{attribute 'GeneratedUsingTerminal: EL6002-0000-0019'}
{attribute addProperty BoxType "EL6002-0000-0019"}
{attribute addProperty Id "StatusAT %I*Status_3D84275F8Data_InAT %I*ARRAY[0..21] OF USINT22"}
{attribute addProperty CRC "1334739266"}
{attribute addProperty Size "30"}
TYPE COM_TxPDO_Map_Inputs_Channel_3801C95E EXTENDS InputBase_8311D824 :
STRUCT
	{attribute addProperty Name "Status"}
	Status AT %I* : Status_3D84275F;
	{attribute addProperty Name "Data_In"}
	Data_In AT %I* : ARRAY[0..21] OF USINT;
END_STRUCT
END_TYPE

(* stored: Version 1.2.0.0, ProductVersion 3.1.4024.9
   DUT COM_TxPDO_Map_Inputs_Channel_3801C95E: Id {32832f36-1ee2-4e00-9320-7c278d393107} *)
